FUNCTION_BLOCK FB_Motoman
VAR_INPUT
	EnableJoystick	: BOOL;
	Value_1	: REAL;
	Value_2	: REAL;
	Value_3	: REAL;
	Value_4	: REAL;
	Value_5	: REAL;
	Value_6	: REAL;	
END_VAR
VAR_IN_OUT
	data	: ST_MotomanIO;	// Raw data from Ethernet/IP
END_VAR
VAR_OUTPUT	
	Error	: UINT;	// 
END_VAR
VAR
	uiDevState: UINT;
	bOk	: BOOL;	
	fbHbTimeout	: TON;
	
	rMaxOutVel : REAL := 1000;

	
	
	pInt	: POINTER TO INT;
	pWord	: POINTER TO WORD;
END_VAR

uiDevState := data.DevState;
// Check comms and heartbeat
bOk := TRUE;	


(*valTemp := LIMIT(-0.6, Value_1, 0.6);

tempLin := F_LIN2(
	X:= valTemp, 
	X1:= -0.6, 
	Y1:= -1000, 
	X2:= 0.6, 
	Y2:= 1000);
	
tempInt := TO_INT(tempLin);

MEMMOVE(ADR(data.out.Vals[0]), ADR(tempInt), 2);
//data.out.Vals[0] := tempInt;
*)

data.out.Vals[0] := PrepareValue(Value_1, rMaxOutVel);
data.out.Vals[1] := PrepareValue(Value_2, rMaxOutVel);
data.out.Vals[2] := PrepareValue(Value_3, rMaxOutVel);

data.out.Cmd.0 := EnableJoystick;

data.out.Cmd.1 := data.out.Vals[0] <> 0 OR data.out.Vals[1] <> 0 OR data.out.Vals[2] <> 0;

IF NOT EnableJoystick THEN 
	MEMSET(ADR(data.out.Cmd), 0, SIZEOF(data.out.Cmd));
	MEMSET(ADR(data.out.Vals), 0, SIZEOF(data.out.Vals));
END_IF
Error := TO_UINT(NOT bOk);

METHOD OpcuaMonitor : BOOL
VAR_INPUT
END_VAR
VAR_IN_OUT
	OpcuaData	: ST_MotomanCtrl;
END_VAR
VAR_OUTPUT
	Error	: BOOL;
END_VAR
VAR_INST
	fbHbMonitor	: FB_HeartbeatMonitor;
	fbBlink	: BLINK;	
	err	: U_OpcuaError;
END_VAR
fbHbMonitor(IN:= OpcuaData.status.input.Heartbeat, PT:= T#2.5S, Q=> );

IF NOT fbHbMonitor.Q THEN
	MEMSET(ADR(OpcuaData.input), 0, SIZEOF(OpcuaData.input));
	Error := TRUE;
ELSE
	Error := FALSE;
END_IF

fbBlink(ENABLE:= TRUE, TIMELOW:= T#500MS, TIMEHIGH:= T#500MS, OUT=> OpcuaData.status.output.Heartbeat);
OpcuaData.status.output.Connected := (THIS^.uiDevState = 0);
END_METHOD

METHOD PrepareValue : INT
VAR_INPUT
	SetVal	: REAL;
	MaxOut	: REAL := 1000;
END_VAR
VAR
	tempWord: WORD;
	tempInt	: INT;
	valTemp: REAL;
	tempLin: REAL;
END_VAR
valTemp := LIMIT(-0.6, SetVal, 0.6);

tempLin := F_LIN2(
	X:= valTemp, 
	X1:= -0.6, 
	Y1:= -MaxOut, 
	X2:= 0.6, 
	Y2:= MaxOut);
	
tempInt := TO_INT(tempLin);

MEMMOVE(ADR(PrepareValue), ADR(tempInt), 2);
END_METHOD

END_FUNCTION_BLOCK

(* stored: Version 1.1.0.1, ProductVersion 3.1.4024.9
   POU FB_Motoman: Id {f0e824e6-1ba2-42aa-8455-a018b9e41f37}, SpecialFunc None
   Method OpcuaMonitor: Id {bc6c407a-71a6-4ae1-8104-4f4653015ad1}
   Method PrepareValue: Id {751eced9-0b6c-4df8-9c73-23da03a5d54e} *)
